# EPICS substitutions: mc05/tpmacApp/Db/pmacStatus.substitutions
file "db/pmacStatus.db"
{
pattern
{SYS,             PMAC,    VERSION  PLC  PORT,  NAXES }
{"XF:16IDB-CT",   "MC:05", "1"      5    "P0",  8     }
}
